Yaskawa INFORM job: sDwell_and_rapid_out_(2).JBI

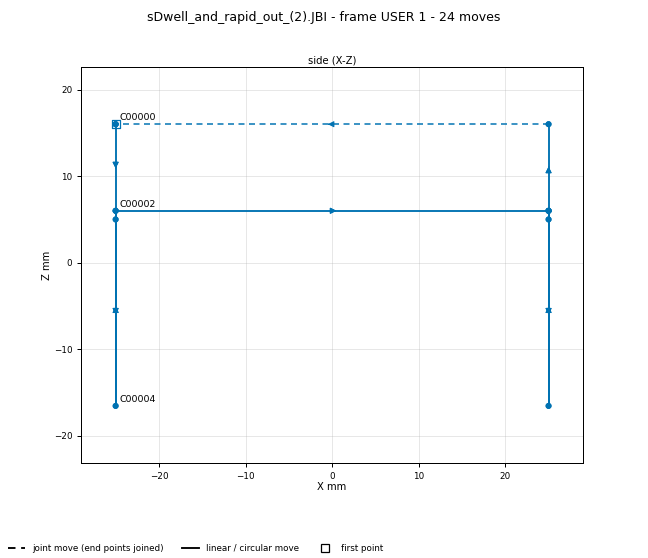
[picture p0: tool path of sDwell_and_rapid_out_(2).JBI in frame USER 1, 24 of 24 moves have a stored position in this frame; points joined in program order, loops and branches not executed]
/JOB
//NAME sDwell_and_rapid_out_(2)
//POS
///NPOS 12,0,0,0,0,0
///USER 1
///TOOL 3
///POSTYPE USER
///RECTAN
///RCONF 1,0,0,0,0,0
C00000=-25.000,10.000,16.000,0.000,-180.000,-30.000
C00001=-25.000,10.000,16.000,0.000,-180.000,-30.000
C00002=-25.000,10.000,6.000,0.000,-180.000,-30.000
C00003=-25.000,10.000,5.000,0.000,-180.000,-30.000
C00004=-25.000,10.000,-16.535,0.000,-180.000,-30.000
C00005=-25.000,10.000,6.000,0.000,-180.000,-30.000
C00006=25.000,10.000,6.000,0.000,-180.000,-30.000
C00007=25.000,10.000,6.000,0.000,-180.000,-30.000
C00008=25.000,10.000,5.000,0.000,-180.000,-30.000
C00009=25.000,10.000,-16.535,0.000,-180.000,-30.000
C00010=25.000,10.000,6.000,0.000,-180.000,-30.000
C00011=25.000,10.000,16.000,0.000,-180.000,-30.000
C00000=-25.000,10.000,16.000,0.000,-180.000,-30.000
C00001=-25.000,10.000,16.000,0.000,-180.000,-30.000
C00002=-25.000,10.000,6.000,0.000,-180.000,-30.000
C00003=-25.000,10.000,5.000,0.000,-180.000,-30.000
C00004=-25.000,10.000,-16.535,0.000,-180.000,-30.000
C00005=-25.000,10.000,6.000,0.000,-180.000,-30.000
C00006=25.000,10.000,6.000,0.000,-180.000,-30.000
C00007=25.000,10.000,6.000,0.000,-180.000,-30.000
C00008=25.000,10.000,5.000,0.000,-180.000,-30.000
C00009=25.000,10.000,-16.535,0.000,-180.000,-30.000
C00010=25.000,10.000,6.000,0.000,-180.000,-30.000
C00011=25.000,10.000,16.000,0.000,-180.000,-30.000
//INST
///ATTR SC,RW,RJ
////FRAME USER 1
///GROUP1 RB1
///LVARS 2,0,0,0,0,0,0,0
NOP
SET LB000 1
SET LB001 25
MOVJ C00000 VJ=17
' Cutting Move Starts
MOVL C00001 V=17 PL=LB000 ACC=LB001 DEC=LB001
MOVL C00002 V=17 PL=LB000 ACC=LB001 DEC=LB001
MOVL C00003 V=17 PL=LB000 ACC=LB001 DEC=LB001
MOVL C00004 V=7 PL=LB000 ACC=LB001 DEC=LB001
MOVL C00005 V=17 PL=LB000 ACC=LB001 DEC=LB001
MOVL C00006 V=17 PL=LB000 ACC=LB001 DEC=LB001
MOVL C00007 V=17 PL=LB000 ACC=LB001 DEC=LB001
MOVL C00008 V=17 PL=LB000 ACC=LB001 DEC=LB001
MOVL C00009 V=7 PL=LB000 ACC=LB001 DEC=LB001
MOVL C00010 V=17 PL=LB000 ACC=LB001 DEC=LB001
' Rapid Move Starts
MOVL C00011 V=17 PL=LB000 ACC=LB001 DEC=LB001
' By Autodesk Fusion CAM 2.0.20494
' Tool = 3
' Spindle = 5000 RPM
' Set Position Level
' Set Acceleration
' Program Start
' First Toolpath Point
' Last Toolpath Point
MOVJ C00000 VJ=17
' Cutting Move Starts
MOVL C00001 V=17 PL=LB000 ACC=LB001 DEC=LB001
MOVL C00002 V=17 PL=LB000 ACC=LB001 DEC=LB001
MOVL C00003 V=17 PL=LB000 ACC=LB001 DEC=LB001
MOVL C00004 V=7 PL=LB000 ACC=LB001 DEC=LB001
MOVL C00005 V=17 PL=LB000 ACC=LB001 DEC=LB001
MOVL C00006 V=17 PL=LB000 ACC=LB001 DEC=LB001
MOVL C00007 V=17 PL=LB000 ACC=LB001 DEC=LB001
MOVL C00008 V=17 PL=LB000 ACC=LB001 DEC=LB001
MOVL C00009 V=7 PL=LB000 ACC=LB001 DEC=LB001
MOVL C00010 V=17 PL=LB000 ACC=LB001 DEC=LB001
' Rapid Move Starts
MOVL C00011 V=17 PL=LB000 ACC=LB001 DEC=LB001
' By Autodesk Fusion CAM 2.0.20494
' Tool = 3
' Spindle = 5000 RPM
' Set Position Level
' Set Acceleration
' Program Start
' First Toolpath Point
END
